// TIA Portal V17 export
// export: Created 2024-08-20T13:37:03.2063023Z, ExportSetting WithDefaults, DisplayName Totally Integrated Automation Portal, DisplayVersion V17 Update 4, DisplayName TIA Portal Openness, DisplayVersion V17 Update 4, DisplayName TIA Portal Version Control Interface, DisplayVersion V17, DisplayName STEP 7 Professional, DisplayVersion V17 Update 4, DisplayName STEP 7 Safety, DisplayVersion V17, DisplayName WinCC Advanced, DisplayVersion V17 Update 4
FUNCTION "AlARME" : Void   // FC3, LAD
{ S7_Optimized_Access := 'TRUE' }
VERSION : 0.1
// stored: AutoNumber true, IsIECCheckEnabled false, SetENOAutomatically false, UDAEnableTagReadback false
BEGIN

REGION Network 1: ALARMES IHM
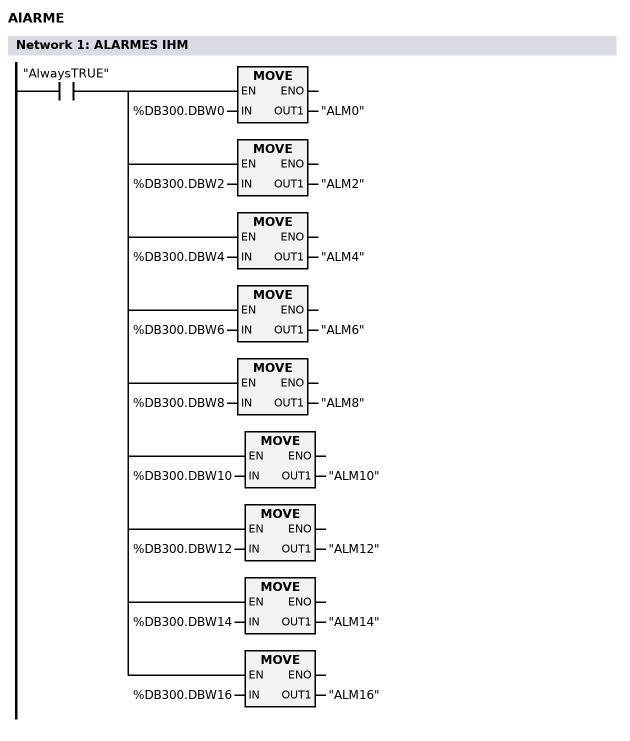
   RUNG wire#powerrail
      Contact( "AlwaysTRUE" )
      wire#w1
      Move(in := %DB300.DBW0, out1 => "ALM0")
   END_RUNG
   RUNG wire#w1
      Move(in := %DB300.DBW2, out1 => "ALM2")
   END_RUNG
   RUNG wire#w1
      Move(in := %DB300.DBW4, out1 => "ALM4")
   END_RUNG
   RUNG wire#w1
      Move(in := %DB300.DBW6, out1 => "ALM6")
   END_RUNG
   RUNG wire#w1
      Move(in := %DB300.DBW8, out1 => "ALM8")
   END_RUNG
   RUNG wire#w1
      Move(in := %DB300.DBW10, out1 => "ALM10")
   END_RUNG
   RUNG wire#w1
      Move(in := %DB300.DBW12, out1 => "ALM12")
   END_RUNG
   RUNG wire#w1
      Move(in := %DB300.DBW14, out1 => "ALM14")
   END_RUNG
   RUNG wire#w1
      Move(in := %DB300.DBW16, out1 => "ALM16")
   END_RUNG
   // the same network as SCL:
   IF "AlwaysTRUE" THEN
       "ALM0" := %DB300.DBW0;
       "ALM2" := %DB300.DBW2;
       "ALM4" := %DB300.DBW4;
       "ALM6" := %DB300.DBW6;
       "ALM8" := %DB300.DBW8;
       "ALM10" := %DB300.DBW10;
       "ALM12" := %DB300.DBW12;
       "ALM14" := %DB300.DBW14;
       "ALM16" := %DB300.DBW16;
   END_IF;
END_REGION
END_FUNCTION
